PROGRAM OverwriteAnalog
VAR
	fbHVACOverwriteAnalog: FB_HVACOverwriteAnalog;
	rValueIn: REAL;
	eCtrlMode: E_HVACCtrlMode;
	rManualValueIn: REAL;
	rValueOut: REAL;
END_VAR

fbHVACOverwriteAnalog(rValueIn:=rValueIn, eCtrlMode:=eCtrlMode, rManualValueIn:=rManualValueIn, rValueOut=>rValueOut);

END_PROGRAM

(* stored: Version 1.1.0.1, ProductVersion 3.1.4024.4
   POU OverwriteAnalog: Id {fc4a1333-6da7-447d-8520-9448d9760879}, SpecialFunc None *)
